Fanuc KAREL source: ABS.kl

PROGRAM T
%NOLOCKGROUP
VAR
 v0 : INTEGER
 res : INTEGER
BEGIN
 res = ABS(v0)
END T
